PROGRAM ConfigDrucksensor
VAR
	state : INT := 1;
	
	(*Daten für die Konfiguration vom Keller-Drucksensor*)	
	UART_akt: 				WORD;
	UARTsettings_akt:		ARRAY[0..1]OF BYTE;
	UARTsettings_neu: 		ARRAY[0..1]OF BYTE  ;//:= [48,0];
	wUARTsettings_neu:		WORD := 0;//:= 112;
	sUARTsettings_neu: 		STRING;
	ModbusRegister:   		Word := 17;
	RegisterLange: 			BYTE := 1;
	ModbusAddress_alt: 		WORD {1..250}:= 1;			//alte Modbusadresse des Slaves. Anfangs gleich der Auslieferungsadresse
	ModbusAddress_neu: 		WORD {3..12} := 11;				//neue Modbusadresse des Slaves. 
	ModbusDataTest: 		DWORD;
	Teststring: 			STRING;
END_VAR

(*Keller-Slaves Konfiguration*)

Teststring:= DWORD_TO_BINSTR(ModbusDataTest,32);

CASE MODBUS.Status_Modbus OF

ConfigPT:

CASE state OF
1:   (* Write Register, write new address to Slave *)	
		IF bConfigPT_setadresse THEN
	 	MODBUS.myModbus.WriteSingleRegister (* writes data to a connected slave. *)
 		(
 		 UnitID:= WORD_TO_BYTE(ModbusAddress_alt),
 		 Quantity:= 1,
 		 MBAddr:= 525,							//Keller: DEV_ADDR 0x020D= DECx525
 		 cbLength:= SIZEOF(ModbusAddress_neu),
 		 pMemoryAddr:= ADR(ModbusAddress_neu),
  		Execute:= TRUE,
  		Timeout:= modbusTimeout,
  		Busy => isModbusBusy,
  		Error => isModbusError,
  		ErrorId => modbusErrorId
  		(* cbRead parameter *));
		
  		IF NOT isModbusBusy THEN
				MODBUS.myModbus.WriteSingleRegister(Execute:= FALSE);
			IF MODBUS.myModbus.Error THEN
				state := 2;
			ELSE
				state := 2;	
			END_IF
		END_IF
		ELSE
			state:= 2;
		END_IF
	
2: 	(* TEST-READ Regs from connected Slave *)

		 MODBUS.myModbus.ReadRegs 
 		(
 		 UnitID:= WORD_TO_BYTE(ModbusAddress_neu),
 		 Quantity:= RegisterLange,						//2 Regs für den Druck P1 oder Temperatur TOB1
 		 MBAddr:= ModbusRegister,						//DECx02 Reg-Adresse für P1, DECx08 Reg-Adresse für TOB1
 		 cbLength:= SIZEOF(ModbusDataTest),
 		 pMemoryAddr:= ADR(ModbusDataTest),
  		Execute:= TRUE,
  		Timeout:= modbusTimeout,
  		Busy => isModbusBusy,
  		Error => isModbusError,
  		ErrorId => modbusErrorId
  		(* cbRead parameter *));
		
  		IF NOT isModbusBusy THEN
				MODBUS.myModbus.ReadRegs(Execute:= FALSE);
			IF myModbus.Error THEN
				state := 2;
			ELSE
				state := 1;	
			END_IF
		END_IF
		
3: (* Write Register, write new UART-settings to Slave *)
	IF bConfigPT_setUART THEN
	 	MODBUS.myModbus.WriteSingleRegister (* writes data to a connected slave. *)
 		(
 		 UnitID:= WORD_TO_BYTE(ModbusAddress_neu),
 		 Quantity:= 1,
 		 MBAddr:= 512,							//Keller: DEV_ADDR 0x020D= DECx525
 		 cbLength:= SIZEOF(wUARTsettings_neu),
 		 pMemoryAddr:= ADR(wUARTsettings_neu),
  		Execute:= TRUE,
  		Timeout:= modbusTimeout,
  		Busy => isModbusBusy,
  		Error => isModbusError,
  		ErrorId => modbusErrorId
  		(* cbRead parameter *));
		
		sUARTsettings_neu:= CONCAT(BYTE_TO_STRING(UARTsettings_neu[1]), BYTE_TO_STRING(UARTsettings_neu[0]));
  		IF NOT isModbusBusy THEN
				MODBUS.myModbus.WriteSingleRegister(Execute:= FALSE);
			IF MODBUS.myModbus.Error THEN
				state := 1;
			ELSE
				state := 4;	
			END_IF
		END_IF
	ELSE
		state:= 4;
  	END_IF

4: (* Read UART-Register from Slave *)

	 	MODBUS.myModbus.ReadRegs
 		(
 		 UnitID:= WORD_TO_BYTE(ModbusAddress_neu),
 		 Quantity:= 1,
 		 MBAddr:= 512,							//Keller: DEV_ADDR 0x020D= DECx525
 		 cbLength:= SIZEOF(UARTsettings_akt),
 		 pMemoryAddr:= ADR(UARTsettings_akt),
  		Execute:= TRUE,
  		Timeout:= modbusTimeout,
  		Busy => isModbusBusy,
  		Error => isModbusError,
  		ErrorId => modbusErrorId
  		(* cbRead parameter *));
		
		//Ändert die Byte-Reihenfolge und konvertiert sie in ein WORT
		UART_akt:= WORD_OF_BYTE(UARTsettings_akt[1], UARTsettings_akt[0]);
		
		
  		IF NOT isModbusBusy THEN
				MODBUS.myModbus.ReadRegs(Execute:= FALSE);
			IF MODBUS.myModbus.Error THEN
				state := 3;
			ELSE
				state := 4;	
			END_IF
		END_IF
		
END_CASE

END_CASE

END_PROGRAM

(* stored: Version 1.1.0.1, ProductVersion 3.1.4019.2
   POU ConfigDrucksensor: Id {b87e714b-b276-4678-8f8f-370ada363745}, SpecialFunc None *)
